// Mitsubishi GX Works2 project: PLC1   PLC: FX3G

// global labels: Global1
VAR_GLOBAL
  startDay AT X007 : BOOL;
  emergency AT X005 : BOOL;
  dayIsWorking AT Y007 : BOOL;
  keepWorking AT Y007 : BOOL;
  PetelStorage AT D1120 : REAL;
  inputPetelStorage AT D1100 : REAL;
  inputLemonStorage AT D1130 : REAL;
  LemonStorage AT D1140 : REAL;
  inputStableizing AT D1150 : REAL;
  stableizing AT D1160 : REAL;
  Lemon AT D1140 : REAL;
  inputLemon AT D1130 : REAL;
  Pete AT D1120 : REAL;
  Petel AT D1120 : REAL;
  inputPetel AT D1100 : REAL;
  inputGummyBears AT D1170 : REAL;
  gummyBears AT D1180 : REAL;
  start_iceCream AT X001 : BOOL;
  iceCreamInput AT D8280 : INT;
END_VAR
VAR_GLOBAL CONSTANT
  divideNum : INT := 400;
END_VAR
VAR_GLOBAL
  iceCreamValue AT D7778 : REAL;
END_VAR
VAR_GLOBAL CONSTANT
  value0 : REAL;
  value5 : REAL := 5;
END_VAR
VAR_GLOBAL
  NURMALiceCream AT M0 : BOOL;
END_VAR
VAR_GLOBAL CONSTANT
  value6 : REAL := 6;
  value10 : REAL := 10;
END_VAR
VAR_GLOBAL
  PINUKiceCream AT M1 : BOOL;
END_VAR
VAR_GLOBAL CONSTANT
  div_400 : REAL := 400;
END_VAR
VAR_GLOBAL
  iceCreamOutput AT D7770 : REAL;
  m_0 AT M0 : BOOL;
  y_11 AT Y011 : BOOL;
  y_10 AT Y010 : BOOL;
  t_200 AT TC200 : BOOL;
END_VAR
VAR_GLOBAL CONSTANT
  sec_5 : INT := 500;
END_VAR
VAR_GLOBAL
  iceCreamMaking AT Y000 : BOOL;
  timer5sec AT TS200 : BOOL;
END_VAR
VAR_GLOBAL CONSTANT
  PetelLimit : REAL := 280;
END_VAR
VAR_GLOBAL
  PetelCheck AT M18 : BOOL;
  LemonCheck AT M21 : BOOL;
  stableizingCheck AT M22 : BOOL;
END_VAR
VAR_GLOBAL CONSTANT
  LemonLimitForNormal : REAL := 35;
  PetelLimitForNormal : REAL := 280;
  stableizingLimitForNormal : REAL := 35;
  petelLimitForPinuk : REAL := 385;
END_VAR
VAR_GLOBAL
  petelCheckPinuk AT M19 : BOOL;
END_VAR
VAR_GLOBAL CONSTANT
  PPLimitNorm : REAL := 280;
END_VAR
VAR_GLOBAL
  PPcheckNorm AT M18 : BOOL;
END_VAR
VAR_GLOBAL CONSTANT
  PLLimitNorm : REAL := 35;
END_VAR
VAR_GLOBAL
  PLCheckNorm AT M19 : BOOL;
END_VAR
VAR_GLOBAL CONSTANT
  PSLimitNorm : REAL := 35;
END_VAR
VAR_GLOBAL
  PSCheckNorm AT M20 : BOOL;
END_VAR
VAR_GLOBAL CONSTANT
  PPLimitPinuk : REAL := 385;
END_VAR
VAR_GLOBAL
  PPCheckPinuk AT M24 : BOOL;
END_VAR
VAR_GLOBAL CONSTANT
  PLLimitPinuk : REAL := 105;
END_VAR
VAR_GLOBAL
  PLCheckPinuk AT M25 : BOOL;
END_VAR
VAR_GLOBAL CONSTANT
  PSLimitPinuk : REAL := 70;
END_VAR
VAR_GLOBAL
  PSCheckPinuk AT M26 : BOOL;
END_VAR
VAR_GLOBAL CONSTANT
  LLLimitNorm : REAL := 420;
END_VAR
VAR_GLOBAL
  LLCheckNorm AT M22 : BOOL;
END_VAR
VAR_GLOBAL CONSTANT
  LSLimitNorm : REAL := 70;
END_VAR
VAR_GLOBAL
  LSCheckNorm AT M21 : BOOL;
END_VAR
VAR_GLOBAL CONSTANT
  LLLimitPinuk : REAL := 560;
END_VAR
VAR_GLOBAL
  LLCheckPinuk AT M27 : BOOL;
  LSCheckPinuk AT M28 : BOOL;
END_VAR
VAR_GLOBAL CONSTANT
  LSLimitPinuk : REAL := 140;
  GLimitNorm : REAL := 28;
END_VAR
VAR_GLOBAL
  GCheckNorm AT M21 : BOOL;
END_VAR
VAR_GLOBAL CONSTANT
  GLimitPinuk : REAL := 70;
END_VAR
VAR_GLOBAL
  GCheckPinuk AT M25 : BOOL;
END_VAR
VAR_GLOBAL CONSTANT
  PLimitNorm : REAL := 280;
END_VAR
VAR_GLOBAL
  PcheckNorm AT M18 : BOOL;
END_VAR
VAR_GLOBAL CONSTANT
  LLimitNorm : REAL := 455;
END_VAR
VAR_GLOBAL
  LCheckNorm AT M19 : BOOL;
END_VAR
VAR_GLOBAL CONSTANT
  SLimitNorm : REAL := 105;
END_VAR
VAR_GLOBAL
  SCheckNorm AT M20 : BOOL;
END_VAR
VAR_GLOBAL CONSTANT
  PLimitPinuk : REAL := 385;
END_VAR
VAR_GLOBAL
  PCheckPinuk AT M22 : BOOL;
END_VAR
VAR_GLOBAL CONSTANT
  LLimitPinuk : REAL := 665;
END_VAR
VAR_GLOBAL
  LCheckPinuk AT M23 : BOOL;
END_VAR
VAR_GLOBAL CONSTANT
  SLimitPinuk : REAL := 210;
END_VAR
VAR_GLOBAL
  SCheckPinuk AT M24 : BOOL;
  NormStart AT M30 : BOOL;
  PinukStart AT M31 : BOOL;
  Normicecream AT M0 : BOOL;
  finish AT M90 : BOOL;
  finishIceCream AT M90 : BOOL;
  startCold AT X002 : BOOL;
END_VAR
VAR_GLOBAL CONSTANT
  Timer8sec : INT := 800;
END_VAR
VAR_GLOBAL
  t_250 AT TC210 : BOOL;
  sec_8 AT TS210 : BOOL;
  isCooling AT Y002 : BOOL;
  temp10 AT X003 : BOOL;
  t_210 AT TC210 : BOOL;
  NoInventory AT M99 : BOOL;
  finishCooling AT M100 : BOOL;
  coolPetel AT D2000 : REAL;
  coolLemon AT D2100 : REAL;
END_VAR
VAR_GLOBAL CONSTANT
  K_350 : REAL := 350;
  K_490 : REAL := 490;
  K_560 : REAL := 560;
  K_700 : REAL := 700;
END_VAR
VAR_GLOBAL
  MIXNorm AT D2200 : REAL;
  MIXPinuk AT D2300 : REAL;
END_VAR
VAR_GLOBAL CONSTANT
  K_868 : REAL := 868;
  K_1330 : REAL := 1330;
END_VAR
VAR_GLOBAL
  finishMIX AT M110 : BOOL;
  hivhuv AT M120 : BOOL;
  hivuv_y5 AT TC2 : BOOL;
END_VAR
VAR_GLOBAL CONSTANT
  blink_time : INT := 5;
END_VAR
VAR_GLOBAL
  ts_2 AT TS2 : BOOL;
  Y_5 AT Y005 : BOOL;
  hivuv_y6 AT TC3 : BOOL;
  ts_3 AT TS3 : BOOL;
  Y_6 AT Y006 : BOOL;
  TC_4 AT TC4 : BOOL;
END_VAR
VAR_GLOBAL CONSTANT
  mixTimeNorm : INT := 30;
END_VAR
VAR_GLOBAL
  TC_5 AT TC5 : BOOL;
END_VAR
VAR_GLOBAL CONSTANT
  mixTimePinuk : WORD := 50;
END_VAR
VAR_GLOBAL
  ts_4 AT TS4 : BOOL;
  ts_5 AT TS5 : BOOL;
  startPacking AT X004 : BOOL;
  packingIsOn AT M111 : BOOL;
  OneGumigam AT CC4 : BOOL;
  OneGumigamStart AT X000 : BOOL;
END_VAR
VAR_GLOBAL CONSTANT
  countOne : INT := 1;
END_VAR
VAR_GLOBAL
  sevenGumigam AT CC5 : BOOL;
END_VAR
VAR_GLOBAL CONSTANT
  count7 : INT := 7;
END_VAR
VAR_GLOBAL
  firstGumigam AT CS4 : BOOL;
  finish7Gumigam AT CS5 : BOOL;
  packingInProcess AT Y004 : BOOL;
  packingIsEnd AT M125 : BOOL;
  TotalPacks AT D1300 : REAL;
END_VAR
VAR_GLOBAL CONSTANT
  addOnePackage : REAL := 1;
END_VAR
VAR_GLOBAL
  updatePackages AT M122 : BOOL;
  packsOutput AT D8282 : INT;
END_VAR
VAR_GLOBAL CONSTANT
  Mul400 : INT := 400;
  Mul40 : INT := 40;
END_VAR
VAR_GLOBAL
  CheckInventory AT M133 : BOOL;
  startCheck AT M135 : BOOL;
END_VAR
VAR_GLOBAL CONSTANT
  ZeroFor8282 : INT;
  ZeroFor1300 : REAL;
END_VAR

// task Task_01 (event TRUE, interval 0, priority 31): POU_01

PROGRAM POU_01
(* structured ladder/FBD written out as ST: instructions are called as NAME(EN, inputs, outputs); _pN, _eN, _tN stand for wires *)
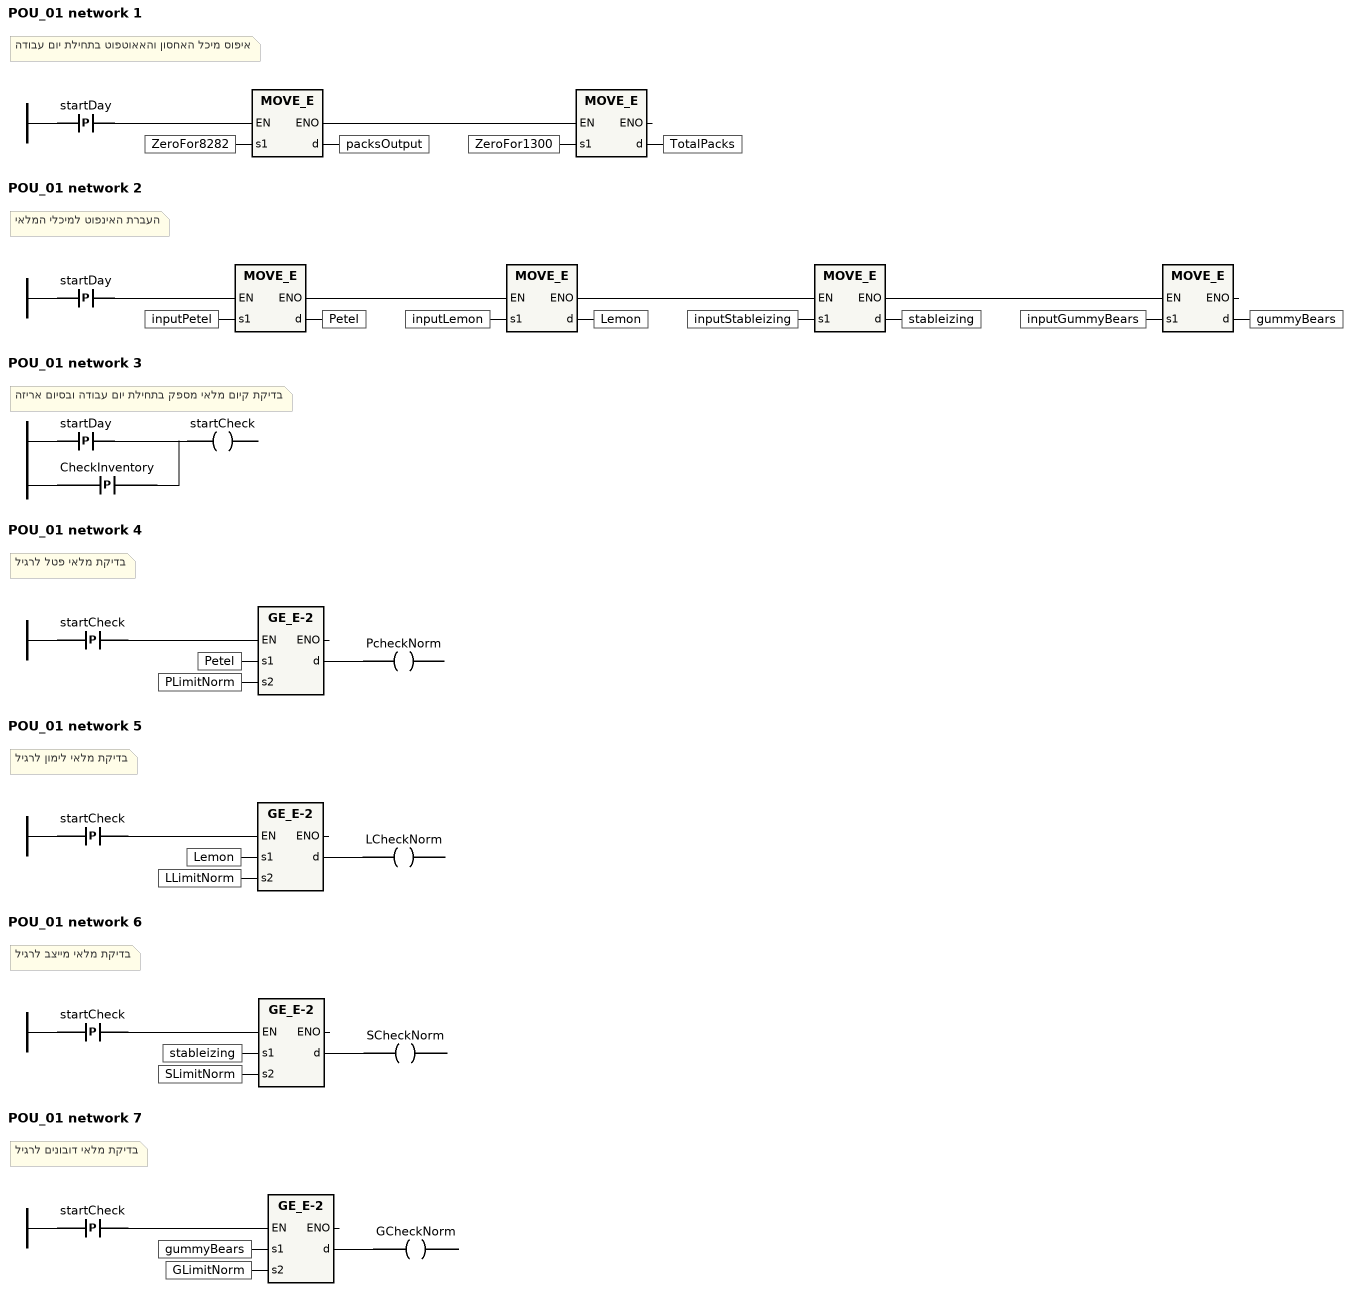
(* network 1 *)
(* איפוס מיכל האחסון והאאוטפוט בתחילת יום עבודה *)
_e1 := MOVE_E(LDP(TRUE, startDay), ZeroFor8282, packsOutput);
MOVE_E(_e1, ZeroFor1300, TotalPacks);
(* network 2 *)
(* העברת האינפוט למיכלי המלאי *)
_e1 := MOVE_E(LDP(TRUE, startDay), inputPetel, Petel);
_e2 := MOVE_E(_e1, inputLemon, Lemon);
_e3 := MOVE_E(_e2, inputStableizing, stableizing);
MOVE_E(_e3, inputGummyBears, gummyBears);
(* network 3 *)
(* בדיקת קיום מלאי מספק בתחילת יום עבודה ובסיום אריזה *)
startCheck := LDP(TRUE, startDay) OR LDP(TRUE, CheckInventory);
(* network 4 *)
(* בדיקת מלאי פטל לרגיל *)
GE_E(LDP(TRUE, startCheck), Petel, PLimitNorm, _t1);
PcheckNorm := _t1;
(* network 5 *)
(* בדיקת מלאי לימון לרגיל *)
GE_E(LDP(TRUE, startCheck), Lemon, LLimitNorm, _t1);
LCheckNorm := _t1;
(* network 6 *)
(* בדיקת מלאי מייצב לרגיל *)
GE_E(LDP(TRUE, startCheck), stableizing, SLimitNorm, _t1);
SCheckNorm := _t1;
(* network 7 *)
(* בדיקת מלאי דובונים לרגיל *)
GE_E(LDP(TRUE, startCheck), gummyBears, GLimitNorm, _t1);
GCheckNorm := _t1;
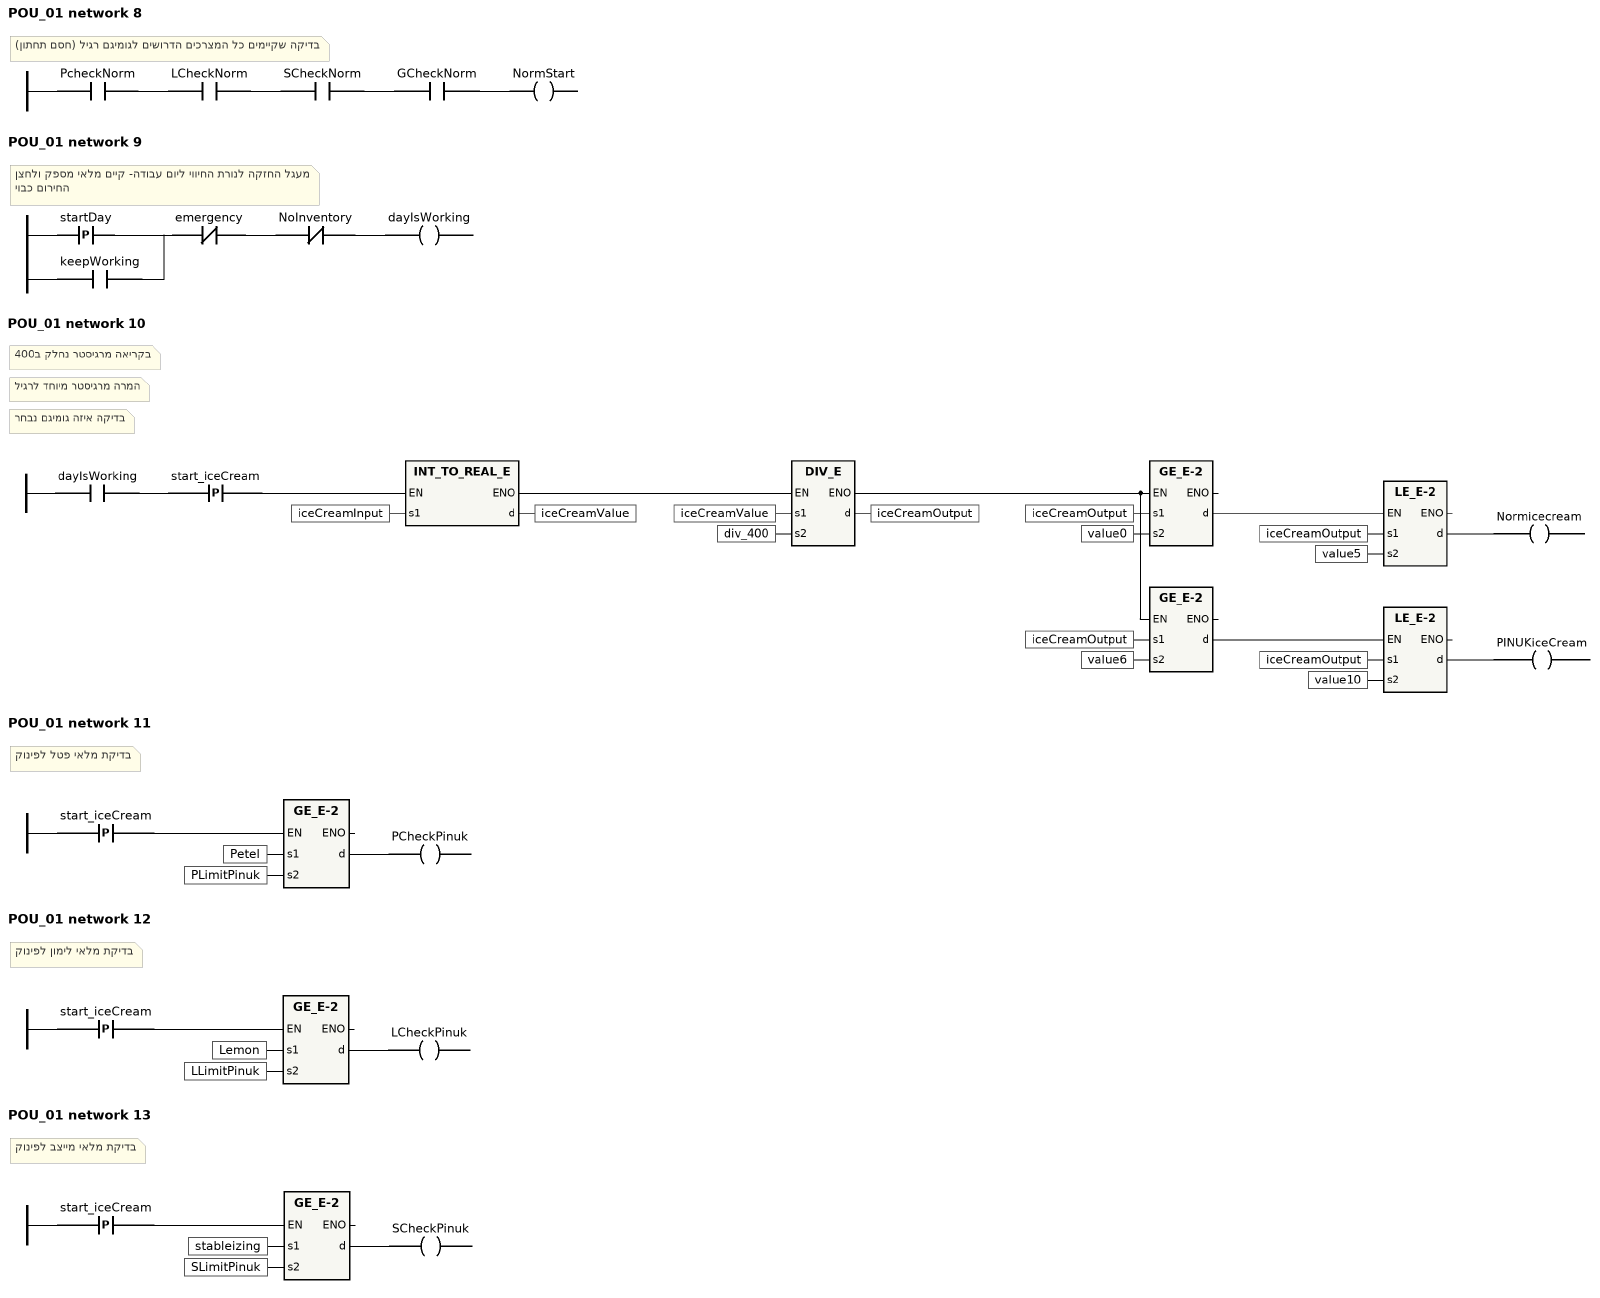
(* network 8 *)
(* בדיקה שקיימים כל המצרכים הדרושים לגומיגם רגיל (חסם תחתון) *)
NormStart := PcheckNorm AND LCheckNorm AND SCheckNorm AND GCheckNorm;
(* network 9 *)
(* מעגל החזקה לנורת החיווי ליום עבודה- קיים מלאי מספק ולחצן החירום כבוי *)
dayIsWorking := ((LDP(TRUE, startDay) OR keepWorking) AND NOT emergency) AND NOT NoInventory;
(* network 10 *)
(* בקריאה מרגיסטר נחלק ב400 *)
(* המרה מרגיסטר מיוחד לרגיל *)
(* בדיקה איזה גומיגם נבחר *)
_e1 := INT_TO_REAL_E(dayIsWorking AND LDP(TRUE, start_iceCream), iceCreamInput, iceCreamValue);
_e2 := DIV_E(_e1, iceCreamValue, div_400, iceCreamOutput);
GE_E(_e2, iceCreamOutput, value0, _t3);
LE_E(_t3, iceCreamOutput, value5, _t4);
Normicecream := _t4;
GE_E(_e2, iceCreamOutput, value6, _t5);
LE_E(_t5, iceCreamOutput, value10, _t6);
PINUKiceCream := _t6;
(* network 11 *)
(* בדיקת מלאי פטל לפינוק *)
GE_E(LDP(TRUE, start_iceCream), Petel, PLimitPinuk, _t1);
PCheckPinuk := _t1;
(* network 12 *)
(* בדיקת מלאי לימון לפינוק *)
GE_E(LDP(TRUE, start_iceCream), Lemon, LLimitPinuk, _t1);
LCheckPinuk := _t1;
(* network 13 *)
(* בדיקת מלאי מייצב לפינוק *)
GE_E(LDP(TRUE, start_iceCream), stableizing, SLimitPinuk, _t1);
SCheckPinuk := _t1;
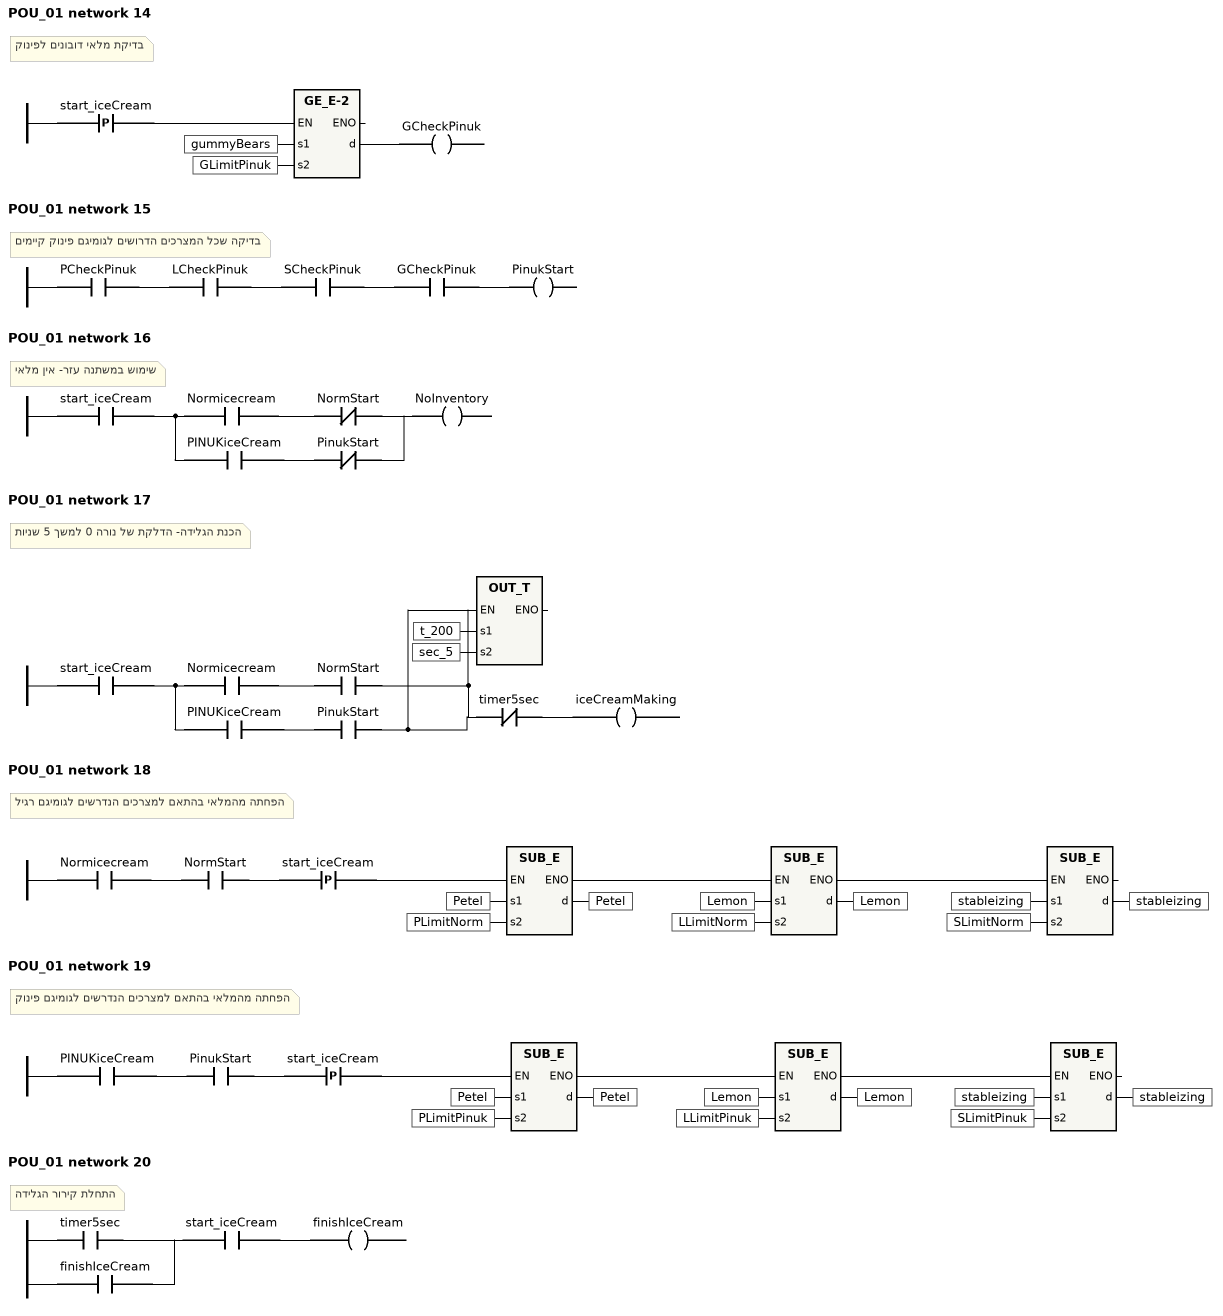
(* network 14 *)
(* בדיקת מלאי דובונים לפינוק *)
GE_E(LDP(TRUE, start_iceCream), gummyBears, GLimitPinuk, _t1);
GCheckPinuk := _t1;
(* network 15 *)
(* בדיקה שכל המצרכים הדרושים לגומיגם פינוק קיימים *)
PinukStart := PCheckPinuk AND LCheckPinuk AND SCheckPinuk AND GCheckPinuk;
(* network 16 *)
(* שימוש במשתנה עזר- אין מלאי *)
NoInventory := (start_iceCream AND Normicecream AND NOT NormStart) OR (start_iceCream AND PINUKiceCream AND NOT PinukStart);
(* network 17 *)
(* הכנת הגלידה- הדלקת של נורה 0 למשך 5 שניות *)
_p1 := (start_iceCream AND Normicecream AND NormStart) OR (start_iceCream AND PINUKiceCream AND PinukStart);
OUT_T(_p1, t_200, sec_5);
iceCreamMaking := _p1 AND NOT timer5sec;
(* network 18 *)
(* הפחתה מהמלאי בהתאם למצרכים הנדרשים לגומיגם רגיל *)
_e1 := SUB_E(Normicecream AND NormStart AND LDP(TRUE, start_iceCream), Petel, PLimitNorm, Petel);
_e2 := SUB_E(_e1, Lemon, LLimitNorm, Lemon);
SUB_E(_e2, stableizing, SLimitNorm, stableizing);
(* network 19 *)
(* הפחתה מהמלאי בהתאם למצרכים הנדרשים לגומיגם פינוק *)
_e1 := SUB_E(PINUKiceCream AND PinukStart AND LDP(TRUE, start_iceCream), Petel, PLimitPinuk, Petel);
_e2 := SUB_E(_e1, Lemon, LLimitPinuk, Lemon);
SUB_E(_e2, stableizing, SLimitPinuk, stableizing);
(* network 20 *)
(* התחלת קירור הגלידה *)
finishIceCream := (timer5sec OR finishIceCream) AND start_iceCream;
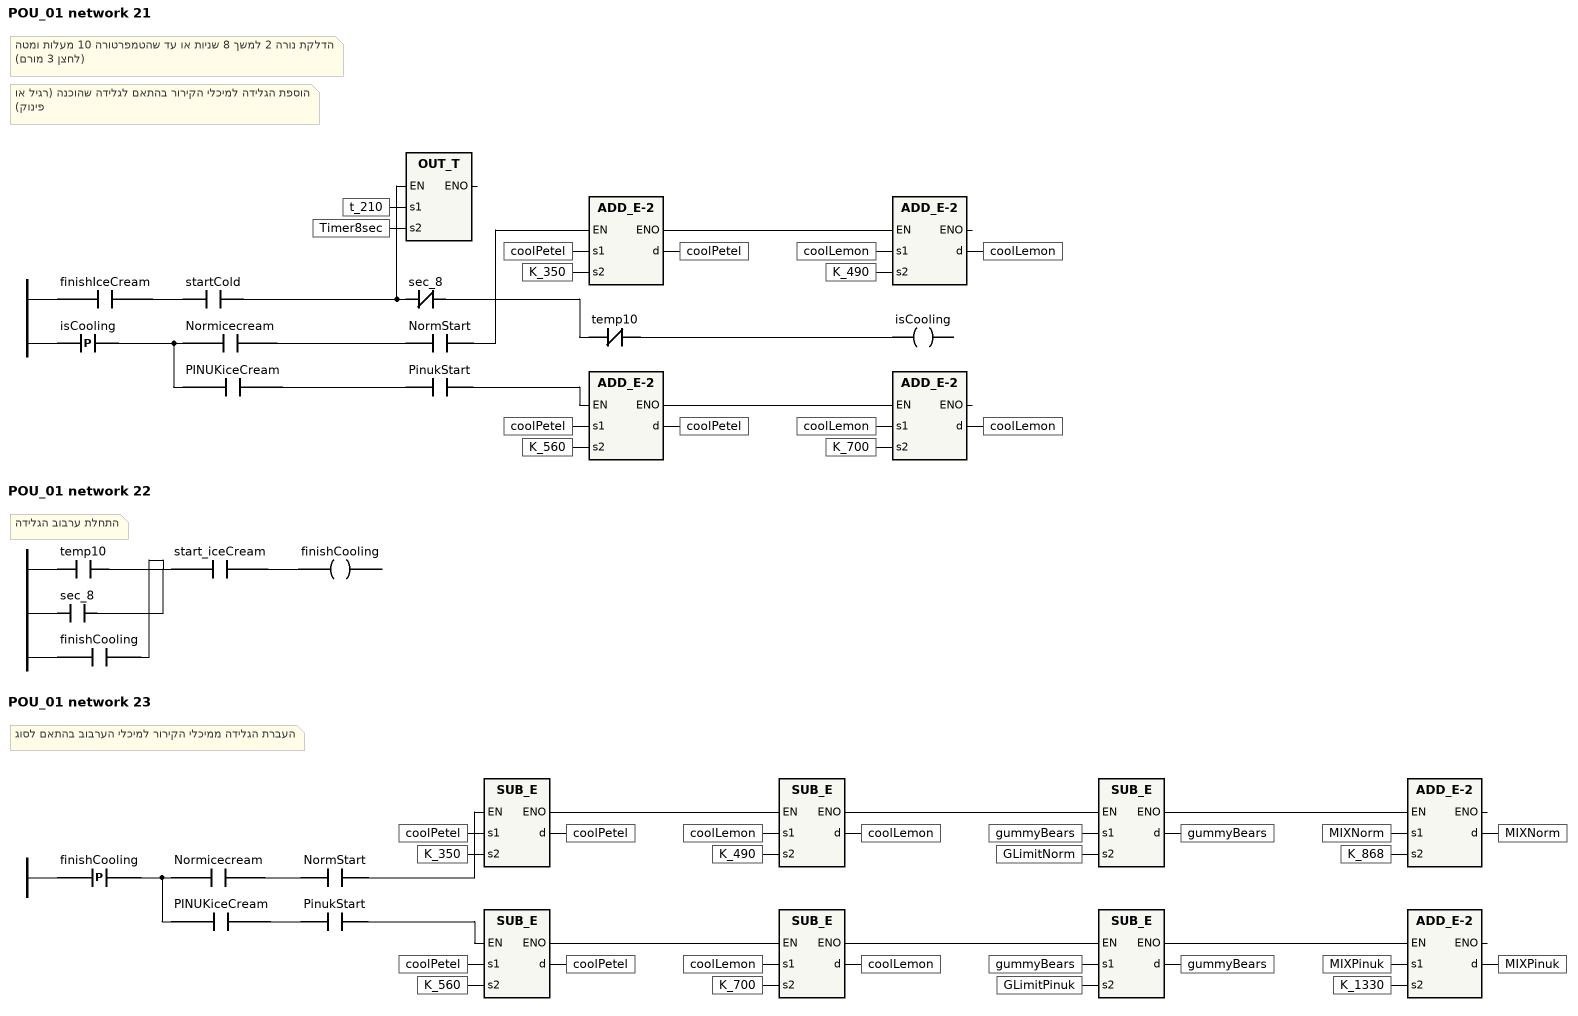
(* network 21 *)
(* הדלקת נורה 2 למשך 8 שניות או עד שהטמפרטורה 10 מעלות ומטה (לחצן 3 מורם) *)
(* הוספת הגלידה למיכלי הקירור בהתאם לגלידה שהוכנה (רגיל או פינוק) *)
_p1 := finishIceCream AND startCold;
OUT_T(_p1, t_210, Timer8sec);
isCooling := _p1 AND NOT sec_8 AND NOT temp10;
_p2 := LDP(TRUE, isCooling);
_e3 := ADD_E(_p2 AND Normicecream AND NormStart, coolPetel, K_350, coolPetel);
ADD_E(_e3, coolLemon, K_490, coolLemon);
_e4 := ADD_E(_p2 AND PINUKiceCream AND PinukStart, coolPetel, K_560, coolPetel);
ADD_E(_e4, coolLemon, K_700, coolLemon);
(* network 22 *)
(* התחלת ערבוב הגלידה *)
finishCooling := (temp10 OR sec_8 OR finishCooling) AND start_iceCream;
(* network 23 *)
(* העברת הגלידה ממיכלי הקירור למיכלי הערבוב בהתאם לסוג *)
_p1 := LDP(TRUE, finishCooling);
_e2 := SUB_E(_p1 AND Normicecream AND NormStart, coolPetel, K_350, coolPetel);
_e3 := SUB_E(_e2, coolLemon, K_490, coolLemon);
_e4 := SUB_E(_e3, gummyBears, GLimitNorm, gummyBears);
ADD_E(_e4, MIXNorm, K_868, MIXNorm);
_e5 := SUB_E(_p1 AND PINUKiceCream AND PinukStart, coolPetel, K_560, coolPetel);
_e6 := SUB_E(_e5, coolLemon, K_700, coolLemon);
_e7 := SUB_E(_e6, gummyBears, GLimitPinuk, gummyBears);
ADD_E(_e7, MIXPinuk, K_1330, MIXPinuk);
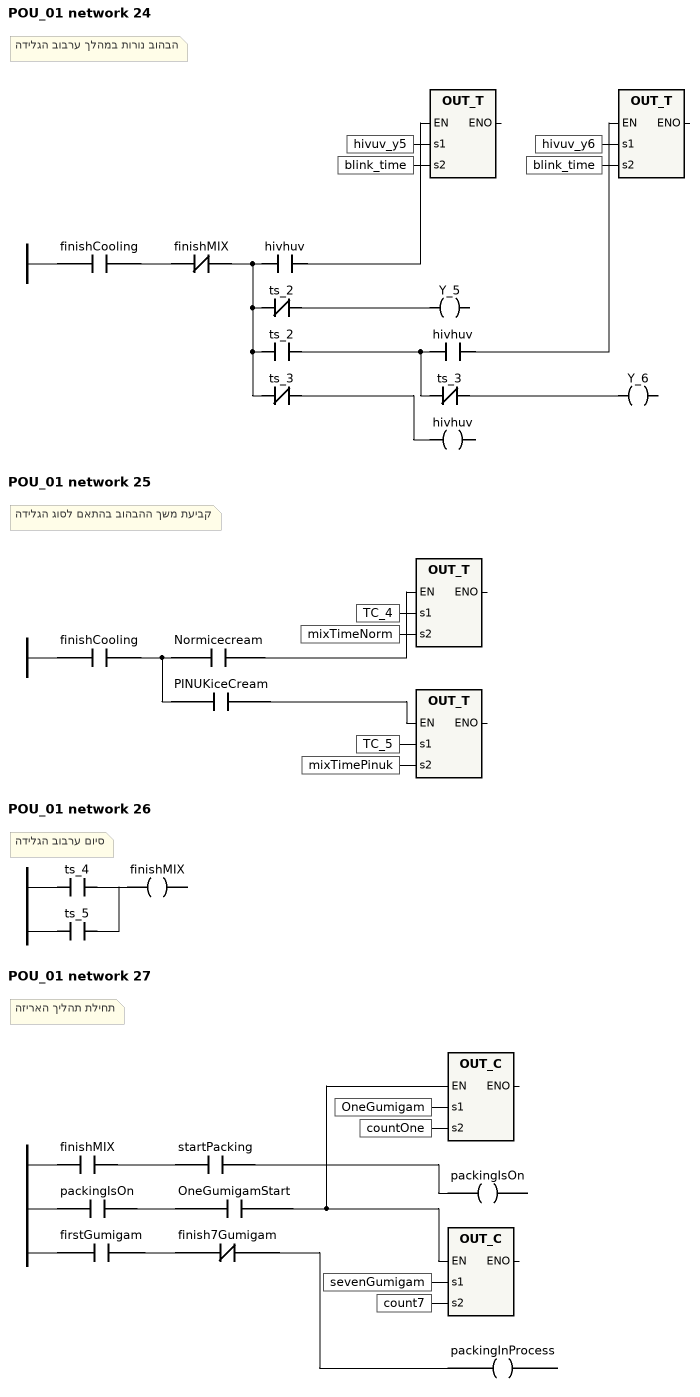
(* network 24 *)
(* הבהוב נורות במהלך ערבוב הגלידה *)
_p1 := finishCooling AND NOT finishMIX;
OUT_T(_p1 AND hivhuv, hivuv_y5, blink_time);
Y_5 := _p1 AND NOT ts_2;
_p2 := _p1 AND ts_2;
OUT_T(_p2 AND hivhuv, hivuv_y6, blink_time);
Y_6 := _p2 AND NOT ts_3;
hivhuv := _p1 AND NOT ts_3;
(* network 25 *)
(* קביעת משך ההבהוב בהתאם לסוג הגלידה *)
OUT_T(finishCooling AND Normicecream, TC_4, mixTimeNorm);
OUT_T(finishCooling AND PINUKiceCream, TC_5, mixTimePinuk);
(* network 26 *)
(* סיום ערבוב הגלידה *)
finishMIX := ts_4 OR ts_5;
(* network 27 *)
(* תחילת תהליך האריזה *)
packingIsOn := finishMIX AND startPacking;
_p1 := packingIsOn AND OneGumigamStart;
OUT_C(_p1, OneGumigam, countOne);
OUT_C(_p1, sevenGumigam, count7);
packingInProcess := firstGumigam AND NOT finish7Gumigam;
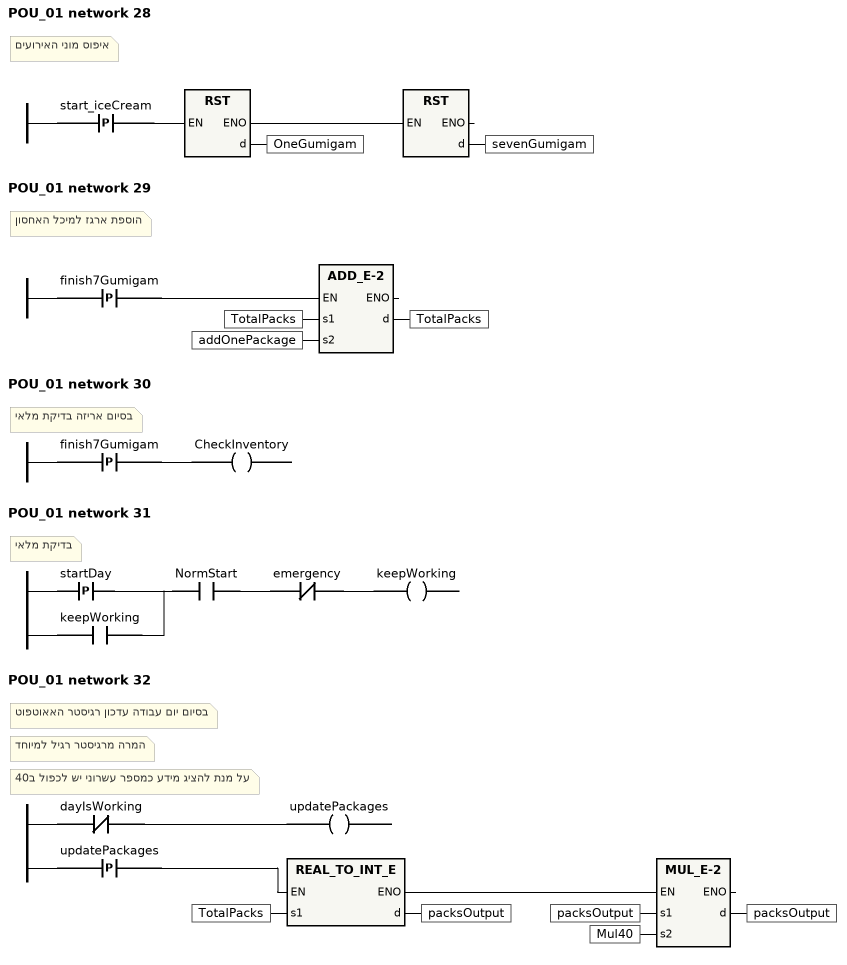
(* network 28 *)
(* איפוס מוני האירועים *)
_e1 := RST(LDP(TRUE, start_iceCream), OneGumigam);
RST(_e1, sevenGumigam);
(* network 29 *)
(* הוספת ארגז למיכל האחסון *)
ADD_E(LDP(TRUE, finish7Gumigam), TotalPacks, addOnePackage, TotalPacks);
(* network 30 *)
(* בסיום אריזה בדיקת מלאי *)
CheckInventory := LDP(TRUE, finish7Gumigam);
(* network 31 *)
(* בדיקת מלאי *)
keepWorking := ((LDP(TRUE, startDay) OR keepWorking) AND NormStart) AND NOT emergency;
(* network 32 *)
(* בסיום יום עבודה עדכון רגיסטר האאוטפוט *)
(* המרה מרגיסטר רגיל למיוחד *)
(* על מנת להציג מידע כמספר עשרוני יש לכפול ב40 *)
updatePackages := NOT dayIsWorking;
_e1 := REAL_TO_INT_E(LDP(TRUE, updatePackages), TotalPacks, packsOutput);
MUL_E(_e1, packsOutput, Mul40, packsOutput);
END_PROGRAM
